PROGRAM MAIN
VAR
END_VAR

END_PROGRAM

(* stored: Version 1.1.0.1
   POU MAIN: Id {9e415983-d2f4-4af7-bce1-9189316ce8d0} *)
